TYPE UNIFIED_PROGRAM_EXECUTED_STEP :
STRUCT
	StepIndex : INT := -1;
	
	Step : REFERENCE TO UNIFIED_PROGRAM_STEP;
END_STRUCT
END_TYPE

(* stored: Version 1.1.0.1
   DUT UNIFIED_PROGRAM_EXECUTED_STEP: Id {1ae1dd06-736e-46a2-a8d0-8bee413aec4d} *)
